// TIA Portal V20 export
FUNCTION "CALL_INIT_FC" : Void   // FC100, LAD
TITLE = Aufruf Initialisierung / Call initialization / Call 初始化
{ S7_Optimized_Access := 'TRUE' }
AUTHOR : Tesla
FAMILY : Base
VERSION : 1.0
// FUNKTIONSBESCHREIBUNG: 
// Der Baustein dient als Aufrufschnittstelle für die Bausteine, die einmalig bzgl. der Initialisierung aufgerufen werden müssen.
// Weitere Hinweise: siehe SICAR anwenderdefinierte Dokumentation / SICAR Online-Hilfe.
// DESCRIPTION OF FUNCTIONS:
// This function is the calling interface for initialization blocks.
// 描述 OF 功能:
// 这个 功能 is  calling 接口 给 初始化 blocks.
// stored: AutoNumber false, SetENOAutomatically false
BEGIN

REGION Network 1: Versorgung Globaler Informationen / Supply global information / 供应 全局 信息
   // 介绍：初始化功能，第一个被调用，调用一次，作用是定义OPMode和HMI数组长度，既最大数量，根据常数来决定。
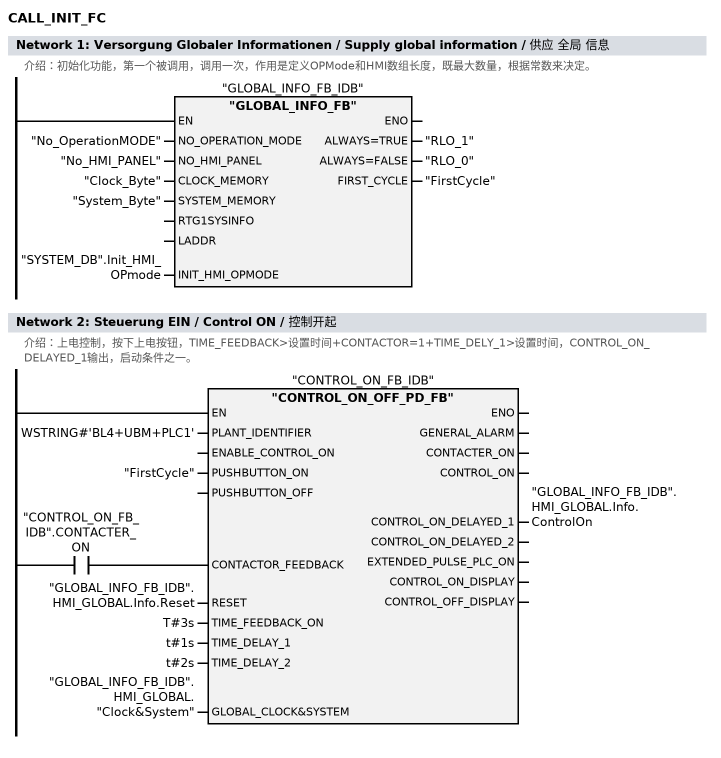
   RUNG wire#powerrail
      "GLOBAL_INFO_FB_IDB"(NO_OPERATION_MODE := "No_OperationMODE", NO_HMI_PANEL := "No_HMI_PANEL", CLOCK_MEMORY := "Clock_Byte", SYSTEM_MEMORY := "System_Byte", RTG1SYSINFO :=, LADDR :=, INIT_HMI_OPMODE := "SYSTEM_DB".Init_HMI_OPmode, "ALWAYS=TRUE" => "RLO_1", "ALWAYS=FALSE" => "RLO_0", FIRST_CYCLE => "FirstCycle")
   END_RUNG
   // the same network as SCL:
   "GLOBAL_INFO_FB_IDB"(NO_OPERATION_MODE := "No_OperationMODE",   // "GLOBAL_INFO_FB"
                        NO_HMI_PANEL := "No_HMI_PANEL",
                        CLOCK_MEMORY := "Clock_Byte",
                        SYSTEM_MEMORY := "System_Byte",
                        INIT_HMI_OPMODE := "SYSTEM_DB".Init_HMI_OPmode,
                        "ALWAYS=TRUE" => "RLO_1",
                        "ALWAYS=FALSE" => "RLO_0",
                        FIRST_CYCLE => "FirstCycle");
END_REGION

REGION Network 2: Steuerung EIN / Control ON / 控制开起
   // 介绍：上电控制，按下上电按钮，TIME_FEEDBACK>设置时间+CONTACTOR=1+TIME_DELY_1>设置时间，CONTROL_ON_DELAYED_1输出，启动条件之一。
   RUNG wire#powerrail
      "CONTROL_ON_FB_IDB"(CONTACTOR_FEEDBACK := wire#w1, PLANT_IDENTIFIER := WSTRING#'BL4+UBM+PLC1', ENABLE_CONTROL_ON :=, PUSHBUTTON_ON := "FirstCycle", PUSHBUTTON_OFF :=, RESET := "GLOBAL_INFO_FB_IDB".HMI_GLOBAL.Info.Reset, TIME_FEEDBACK_ON := T#3s, TIME_DELAY_1 := t#1s, TIME_DELAY_2 := t#2s, "GLOBAL_CLOCK&SYSTEM" := "GLOBAL_INFO_FB_IDB".HMI_GLOBAL."Clock&System", GENERAL_ALARM =>, CONTACTER_ON =>, CONTROL_ON =>, CONTROL_ON_DELAYED_1 => "GLOBAL_INFO_FB_IDB".HMI_GLOBAL.Info.ControlOn, CONTROL_ON_DELAYED_2 =>, EXTENDED_PULSE_PLC_ON =>, CONTROL_ON_DISPLAY =>, CONTROL_OFF_DISPLAY =>)
   END_RUNG
   RUNG wire#powerrail
      Contact( "CONTROL_ON_FB_IDB".CONTACTER_ON )
   END_RUNG wire#w1
   // the same network as SCL:
   "CONTROL_ON_FB_IDB"(PLANT_IDENTIFIER := WSTRING#'BL4+UBM+PLC1',   // "CONTROL_ON_OFF_PD_FB"
                       PUSHBUTTON_ON := "FirstCycle",
                       CONTACTOR_FEEDBACK := "CONTROL_ON_FB_IDB".CONTACTER_ON,
                       RESET := "GLOBAL_INFO_FB_IDB".HMI_GLOBAL.Info.Reset,
                       TIME_FEEDBACK_ON := T#3s,
                       TIME_DELAY_1 := t#1s,
                       TIME_DELAY_2 := t#2s,
                       "GLOBAL_CLOCK&SYSTEM" := "GLOBAL_INFO_FB_IDB".HMI_GLOBAL."Clock&System",
                       CONTROL_ON_DELAYED_1 => "GLOBAL_INFO_FB_IDB".HMI_GLOBAL.Info.ControlOn);
END_REGION
END_FUNCTION
